FUNCTION_BLOCK Generator
  (* Standard: 61499-2 *)
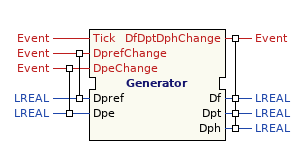
  EVENT_INPUT
    Tick;
    DprefChange WITH Dpref;
    DpeChange WITH Dpe;
  END_EVENT
  EVENT_OUTPUT
    DfDptDphChange WITH Df, Dpt, Dph;
  END_EVENT
  VAR_INPUT
    Dpref : LREAL;
    Dpe : LREAL := 0.1;
  END_VAR
  VAR_OUTPUT
    Df : LREAL;
    Dpt : LREAL;
    Dph : LREAL;
  END_VAR
  VAR
    StepSize : LREAL := 0.0001;
    Kh : LREAL := 1.0;
    Kt : LREAL := 1.0;
    Kp : LREAL := 120;
    Th : LREAL := 0.08;
    Tt : LREAL := 0.3;
    Tp : LREAL := 20;
    R : LREAL := 2.4;
  END_VAR
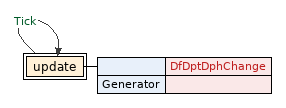
  EC_STATES
    update : -> DfDptDphChange, Generator;
  END_STATES
  EC_TRANSITIONS
    update TO update := Tick;
  END_TRANSITIONS
  ALGORITHM Generator IN ST:
		Dph := Dph + ((Kh * Dpref - (Kh * Df)/R - Dph) / Th) * StepSize;
        if Dph > 0.15 then
            Dph := 0.15;
        elsif Dph < -0.15 then
            Dph := -0.15;
        end_if;
		Dpt := Dpt + ((Kt * Dph - Dpt) / Tt) * StepSize;
        Df := Df + ((Kp * Dpt - Kp * Dpe - Df) / Tp) * StepSize;
  END_ALGORITHM
END_FUNCTION_BLOCK
